TYPE ST_OverCurrProtection_HWQ :
STRUCT
  bCtrlResetCh1   : BOOL;
  bCtrlSwitchCh1  : BOOL;
  bCtrlResetCh2   : BOOL;
  bCtrlSwitchCh2  : BOOL;
END_STRUCT
END_TYPE

(* stored: Version 1.1.0.1, ProductVersion 3.1.4024.12
   DUT ST_OverCurrProtection_HWQ: Id {7bbb8374-8ae1-4712-a7a1-0be615895038} *)
